(* CODESYS project Elevator - Project Code.project

Project tree, tasks and I/O mapping:
  Device : CODESYS Control Win V3, 3S - Smart Software Solutions GmbH, version 3.5.16.20
    application Application
      libraries: Standard, * (System)
      task MainTask (cyclic, interval t#20ms, priority 1) calls Simulation
      task VISU_TASK (cyclic, interval 100 ms, priority 31) calls VisuElems.Visu_Prg
      global variables GVL
      visualisation Visualization
      program Simulation [ST]
  text list GlobalTextList
*)

// Device/Application/GVL
{attribute 'qualified_only'}
VAR_GLOBAL
(* Elevator managing variables*)
	Open: BOOL;				(* Sensor: the door is fully open*)
	Closed: BOOL;			(* Sensor: the door is fully closed*)
	LimitDown: BOOL;		(* Sensor: lower limit sensor, if TRUE the lift has reached the lower limit*)
	LimitUp: BOOL;			(* Sensor: upper limit sensor, if TRUE the lift has reached the upper limit*)
	DeckSensor: BOOL;		(* Sensor: if TRUE the cab is in proximity of a deck*)
	RampSensor: BOOL;		(* Sensor: if TRUE the cab is in proximity of a ramp*)
	Presence :BOOL; 		(* Sensor: if TRUE something blocks the door photocell*)
	Emergency: BOOL;		(* Input: if TRUE the emergency button has been pressed*)

	Closing: BOOL;			(* Actuator: if TRUE the door starts closing*)
	Opening: BOOL;			(* Actuator: the door starts opening*)
	Motor_on: BOOL;			(* Actuator: if TRUE the lift pulley motor start moving*)
	Up: BOOL;				(* Actuator parameter: if TRUE the lift moves upward, downward otherwise*)
	Vel: BOOL;				(* Actuator parameter: motor speed, if TRUE high speed, low speed otherwise*)


	Current: INT;  			(* Visualization: variable used to storage the current deck*)
    Destination: INT;		(* Visualization: variable used to storage the the destination deck*)
	EmergencyVis: BOOL; 	(* Visualization: if TRUE the emergency light is turned on*)

	InitialDeck: INT := 1;	(* Only for simulation: variable used to define the initial deck*)
	InitCycle: BOOL := FALSE;(* Only for simulation: used to execute the instruction at the first cycle*)
	Height: INT;			(* Only for simulation: elevator height*)
	DeckRest: INT;        	(* Only for simulation: division rest for generating deck sensor*)
	Memory: INT;
	RampRest: INT;			(* Only for simulation: division rest for generating the ramp position*)
	MemoryR: INT;
	Door: INT;				(* Only for simulation: to visualize the closing of the door*)
	Displacement: INT;		(* Only for simulation: lift displacement, dependent on the motor speed*)

 (*Inputs: internal panel variables*)
	PG: BOOL;
	P1: BOOL;
	P2: BOOL;
	P3: BOOL;
	P4: BOOL;
	P5: BOOL;
	P6: BOOL;
	P7: BOOL;

(*Visualization: internal panel variables used to turn on the LED*)
	PGVis: BOOL;
	P1Vis: BOOL;
	P2Vis: BOOL;
	P3Vis: BOOL;
	P4Vis: BOOL;
	P5Vis: BOOL;
	P6Vis: BOOL;
	P7Vis: BOOL;

(*Inputs: external panel variables*)
	UpDeckG: BOOL;
	UpDeck1: BOOL;
	UpDeck2: BOOL;
	UpDeck3: BOOL;
	UpDeck4: BOOL;
	UpDeck5: BOOL;
	UpDeck6: BOOL;
	DownDeck7: BOOL;
	DownDeck6: BOOL;
	DownDeck5: BOOL;
	DownDeck4: BOOL;
	DownDeck3: BOOL;
	DownDeck2: BOOL;
	DownDeck1: BOOL;

(*Visualization: external panel variables used to turn on the LED*)
	UpDeckGVis: BOOL;
	UpDeck1Vis: BOOL;
	UpDeck2Vis: BOOL;
	UpDeck3Vis: BOOL;
	UpDeck4Vis: BOOL;
	UpDeck5Vis: BOOL;
	UpDeck6Vis: BOOL;
	DownDeck7Vis: BOOL;
	DownDeck6Vis: BOOL;
	DownDeck5Vis: BOOL;
	DownDeck4Vis: BOOL;
	DownDeck3Vis: BOOL;
	DownDeck2Vis: BOOL;
	DownDeck1Vis: BOOL;

(*Only for simulation: variables used to simulate the fault on deck sensor*)
	SensorG: BOOL;				(* if TRUE the magnetic information for deck G is lost and the deck sensor cannot become TRUE*)
	Sensor1: BOOL;				(* if TRUE the magnetic information for deck 1 is lost and the deck sensor cannot become TRUE*)
	Sensor2: BOOL;
	Sensor3: BOOL;
	Sensor4: BOOL;
	Sensor5: BOOL;
	Sensor6: BOOL;
	Sensor7: BOOL;
	FaultSensorAlarm: BOOL; 	(* Visulaization: if TRUE alerts the user of a deck sensor fault*)

(*Only for simulation: variables used to simulate the fault on ramp sensor*)
	RampGUp: BOOL;
	Ramp1Down: BOOL;
	Ramp1Up:BOOL;
	Ramp2Down: BOOL;
	Ramp2Up:BOOL;
	Ramp3Down: BOOL;
	Ramp3Up:BOOL;
	Ramp4Down: BOOL;
	Ramp4Up:BOOL;
	Ramp5Down: BOOL;
	Ramp5Up:BOOL;
	Ramp6Down: BOOL;
	Ramp6Up:BOOL;
	Ramp7Down: BOOL;
	FaultRampAlarm: BOOL; 		(* Visulaization: if TRUE alerts the user of a ramp sensor fault*)
	SensorGOK: BOOL;
	Sensor1OK: BOOL;
	Sensor2OK: BOOL;
	Sensor6OK: BOOL;
	Sensor3OK: BOOL;
	Sensor4OK: BOOL;
	Sensor5OK: BOOL;
	Sensor7OK: BOOL;
	RampGUpOK: BOOL;
	Ramp1DownOK: BOOL;
	Ramp1UpOK: BOOL;
	Ramp2DownOK: BOOL;
	Ramp2UpOK: BOOL;
	Ramp3DownOK: BOOL;
	Ramp3UpOK: BOOL;
	Ramp4DownOK: BOOL;
	Ramp4UpOK: BOOL;
	Ramp5DownOK: BOOL;
	Ramp5UpOK: BOOL;
	Ramp6DownOK: BOOL;
	Ramp6UpOK: BOOL;
	Ramp7DownOK: BOOL;
	Ramp7UpOK: BOOL;
END_VAR

// Device/Application/Simulation
PROGRAM Simulation
VAR
END_VAR

(* Initial position of the cab inside the hoistway. It is executed only at the first cycle.  *)
IF NOT GVL.InitCycle THEN
			GVL.InitCycle := TRUE ;
			GVL.Height := 20 * GVL.InitialDeck;
		    GVL.Door := 0;
			GVL.Current := GVL.Height / 20;
END_IF;

(* Elevator management, these instructions are executed each cycle time*)

(* Elevator door control. *)
IF GVL.Closing THEN
	GVL.Door := GVL.Door + 1;		(*Closing door management*)
	GVL.Open := FALSE;
END_IF

IF GVL.Door >= 60 THEN						(* Closed door limit*)
	GVL.Closed := TRUE;
END_IF

IF GVL.Opening THEN
	GVL.Door := GVL.Door - 1; 	(* Opening door management*)
	GVL.Closed := FALSE;
END_IF

IF GVL.Door <= 0 THEN							(* Open door limit*)
	GVL.Open := TRUE;
END_IF


(* Maximum and minimum management in the door simulation*)
IF GVL.Door < 0 THEN
	 GVL.Door := 0;
END_IF

IF GVL.Door > 60 THEN
	GVL.Door := 60;
END_IF


(* Control of the cab position inside the hostway. *)
(* Displacement definition for graphic visualization*)
IF GVL.Vel THEN 
	GVL.Displacement := 2;
ELSE 
	GVL.Displacement := 1;
END_IF


(* Height modification relying on direction and speed*)
IF GVL.Motor_on AND GVL.Up THEN
	GVL.Height := GVL.Height + GVL.Displacement;
	GVL.LimitDown := FALSE;
END_IF

IF GVL.Motor_on AND NOT GVL.Up THEN
	GVL.Height := GVL.Height - GVL.Displacement;
	GVL.LimitUp := FALSE;
END_IF


(* Limits for visualization*)
IF GVL.Height < -20 THEN
	GVL.Height := -20;
END_IF

IF GVL.Height > 160 THEN
	GVL.Height := 160;
END_IF

(* Limit sensors management*)
IF GVL.Height <= -10 THEN
	GVL.LimitDown := TRUE;
END_IF

IF GVL.Height >= 150 THEN
	 GVL.LimitUp := TRUE;
END_IF


(*-------------------------------------------------------------------*)
(*  Fault Management (Deck and Ramp Sensors)   *)
(*-------------------------------------------------------------------*)
(* Deck Sensor*)
(* Range of value where the deck sensor is active*)
IF ((GVL.Height >= -1) AND (GVL.Height <= 1)) THEN
	GVL.SensorGOK := TRUE;
ELSE  
	GVL.SensorGOK := FALSE;
END_IF

IF ((GVL.Height >= 20-1) AND (GVL.Height <= 20+1)) THEN
	GVL.Sensor1OK := TRUE;
ELSE  
	GVL.Sensor1OK := FALSE;
END_IF

IF ((GVL.Height >= 40-1) AND (GVL.Height <= 40+1)) THEN
	GVL.Sensor2OK := TRUE;
ELSE  
	GVL.Sensor2OK := FALSE;
END_IF

IF ((GVL.Height >= 60-1) AND (GVL.Height <= 60+1)) THEN
	GVL.Sensor3OK := TRUE;
ELSE  
	GVL.Sensor3OK := FALSE;
END_IF

IF ((GVL.Height >= 80-1) AND (GVL.Height <= 80+1)) THEN
	GVL.Sensor4OK := TRUE;
ELSE  
	GVL.Sensor4OK := FALSE;
END_IF

IF ((GVL.Height >= 100-1) AND (GVL.Height <= 100+1)) THEN
	GVL.Sensor5OK := TRUE;
ELSE   
	GVL.Sensor5OK := FALSE;
END_IF

IF ((GVL.Height >= 120-1) AND (GVL.Height <= 120+1)) THEN
	GVL.Sensor6OK := TRUE;
ELSE  
	GVL.Sensor6OK := FALSE;
END_IF

IF ((GVL.Height >= 140-1) AND (GVL.Height <= 140+1)) THEN
	GVL.Sensor7OK := TRUE;
ELSE  
	GVL.Sensor7OK := FALSE;
END_IF

GVL.DeckSensor := (GVL.SensorGOK AND NOT GVL.SensorG) OR
				    (GVL.Sensor1OK AND NOT GVL.Sensor1) OR
				    (GVL.Sensor2OK AND NOT GVL.Sensor2) OR
				    (GVL.Sensor3OK AND NOT GVL.Sensor3) OR
				    (GVL.Sensor4OK AND NOT GVL.Sensor4) OR
				    (GVL.Sensor5OK AND NOT GVL.Sensor5) OR
				    (GVL.Sensor6OK AND NOT GVL.Sensor6) OR
				    (GVL.Sensor7OK AND NOT GVL.Sensor7);

(* Ramp Sensor*)
(* Range of value where the ramp sensor is active*)
IF ((GVL.Height >= 5-1) AND (GVL.Height <= 5+1)) THEN
	GVL.RampGUpOK := TRUE;
ELSE 
	GVL.RampGUpOK := FALSE;
END_IF

(* Ramp close to deck 1*)
IF ((GVL.Height >= 15-1) AND (GVL.Height <= 15+1)) THEN
	GVL.Ramp1DownOK := TRUE;
ELSE 
	GVL.Ramp1DownOK := FALSE;
END_IF

IF ((GVL.Height >= 25-1) AND (GVL.Height <= 25+1)) THEN
	GVL.Ramp1UpOK := TRUE;
ELSE 
	GVL.Ramp1UpOK := FALSE;
END_IF

(* Ramp close to deck 2*)
IF ((GVL.Height >= 35-1) AND (GVL.Height <= 35+1)) THEN
	GVL.Ramp2DownOK := TRUE;
ELSE 
	GVL.Ramp2DownOK := FALSE;
END_IF

IF ((GVL.Height >= 45-1) AND (GVL.Height <= 45+1)) THEN
	GVL.Ramp2UpOK := TRUE;
ELSE 
	GVL.Ramp2UpOK := FALSE;
END_IF

(*Ramp close to deck  3*)
IF ((GVL.Height >= 55-1) AND (GVL.Height <= 55+1)) THEN
	GVL.Ramp3DownOK := TRUE;
ELSE 
	GVL.Ramp3DownOK := FALSE;
END_IF

IF ((GVL.Height >= 65-1) AND (GVL.Height <= 65+1)) THEN
	GVL.Ramp3UpOK := TRUE;
ELSE 
	GVL.Ramp3UpOK := FALSE;
END_IF

(* Ramp close to deck  4*)
IF ((GVL.Height >= 75-1) AND (GVL.Height <= 75+1)) THEN
	GVL.Ramp4DownOK := TRUE;
ELSE 
	GVL.Ramp4DownOK := FALSE;
END_IF

IF ((GVL.Height >= 85-1) AND (GVL.Height <= 85+1)) THEN
	GVL.Ramp4UpOK := TRUE;
ELSE 
	GVL.Ramp4UpOK:=FALSE;
END_IF

(* Ramp close to deck  5*)
IF ((GVL.Height >= 95-1) AND (GVL.Height <= 95+1)) THEN
	GVL.Ramp5DownOK := TRUE;
ELSE 
	GVL.Ramp5DownOK := FALSE;
END_IF

IF ((GVL.Height >= 105-1) AND (GVL.Height <= 105+1)) THEN
	GVL.Ramp5UpOK := TRUE;
ELSE
	GVL.Ramp5UpOK := FALSE;
END_IF

(* Ramp close to deck  6*)
IF ((GVL.Height >= 115-1) AND (GVL.Height <= 115+1)) THEN
	GVL.Ramp6DownOK := TRUE;
ELSE 
	GVL.Ramp6DownOK := FALSE;
END_IF

IF ((GVL.Height >= 125-1) AND (GVL.Height <= 125+1)) THEN
	GVL.Ramp6UpOK := TRUE;
ELSE 
	GVL.Ramp6UpOK := FALSE;
END_IF

(* Ramp close to deck  7*)
IF ((GVL.Height >= 135-1) AND (GVL.Height <= 135+1)) THEN
	GVL.Ramp7DownOK := TRUE;
ELSE 
	GVL.Ramp7DownOK := FALSE;
END_IF

GVL.RampSensor:=(GVL.RampGUpOK AND NOT GVL.RampGUp) OR 
								(GVL.Ramp1DownOK AND NOT GVL.Ramp1Down ) OR 
								(GVL.Ramp1UpOK AND NOT GVL.Ramp1Up ) OR
								(GVL.Ramp2DownOK AND NOT GVL.Ramp2Down ) OR 
								(GVL.Ramp2UpOK AND NOT GVL.Ramp2Up ) OR
								(GVL.Ramp3DownOK AND NOT GVL.Ramp3Down ) OR
 								(GVL.Ramp3UpOK AND NOT GVL.Ramp3Up ) OR
								(GVL.Ramp4DownOK AND NOT GVL.Ramp4Down ) OR
 								(GVL.Ramp4UpOK AND NOT GVL.Ramp4Up ) OR
								(GVL.Ramp5DownOK AND NOT GVL.Ramp5Down ) OR
 								(GVL.Ramp5UpOK AND NOT GVL.Ramp5Up ) OR
								(GVL.Ramp6DownOK AND NOT GVL.Ramp6Down ) OR
								(GVL.Ramp6UpOK AND NOT GVL.Ramp6Up ) OR
								(GVL.Ramp7DownOK AND NOT GVL.Ramp7Down );

END_PROGRAM

// Device/Application/Visualization
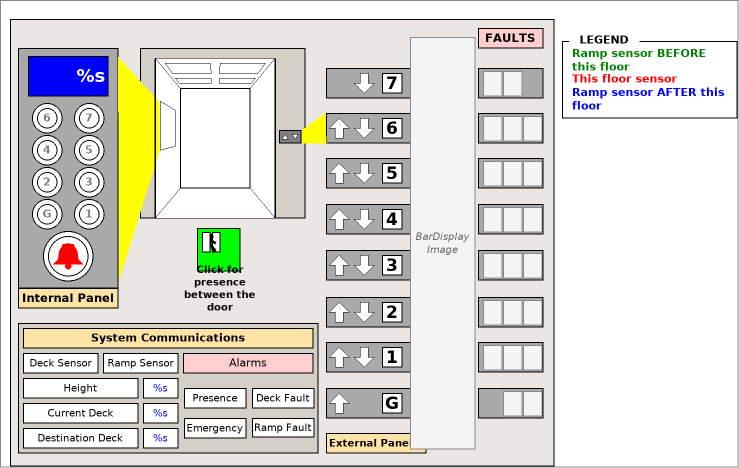
VISUALIZATION Visualization  // 739x468
    Rectangle (10,19 544x447)
    Rectangle (197,228 43x43), colour toggle: GVL.Presence
    Rectangle (18,323 300x130)
    Rectangle (326,433 100x20), "External Panels"
    Rectangle (326,342 100x30)
    Rectangle (382,347 20x20), "1"
    Polygon (354,357) (360,357) (360,347) (368,347) (368,357) (374,357) (364,367), colour toggle: GVL.DownDeck1Vis
        tap GVL.DownDeck1
    Polygon (329,357) (335,357) (335,367) (343,367) (343,357) (349,357) (339,347), colour toggle: GVL.UpDeck1Vis
        tap GVL.UpDeck1
    Rectangle (326,297 100x30)
    Rectangle (382,302 20x20), "2"
    Polygon (354,312) (360,312) (360,302) (368,302) (368,312) (374,312) (364,322), colour toggle: GVL.DownDeck2Vis
        tap GVL.DownDeck2
    Polygon (329,312) (335,312) (335,322) (343,322) (343,312) (349,312) (339,302), colour toggle: GVL.UpDeck2Vis
        tap GVL.UpDeck2
    Rectangle (326,250 100x30)
    Rectangle (382,255 20x20), "3"
    Polygon (354,265) (360,265) (360,255) (368,255) (368,265) (374,265) (364,275), colour toggle: GVL.DownDeck3Vis
        tap GVL.DownDeck3
    Polygon (329,265) (335,265) (335,275) (343,275) (343,265) (349,265) (339,255), colour toggle: GVL.UpDeck3Vis
        tap GVL.UpDeck3
    Rectangle (326,204 100x30)
    Rectangle (382,209 20x20), "4"
    Polygon (354,219) (360,219) (360,209) (368,209) (368,219) (374,219) (364,229), colour toggle: GVL.DownDeck4Vis
        tap GVL.DownDeck4
    Polygon (329,219) (335,219) (335,229) (343,229) (343,219) (349,219) (339,209), colour toggle: GVL.UpDeck4Vis
        tap GVL.UpDeck4
    Rectangle (326,158 100x30)
    Rectangle (382,163 20x20), "5"
    Polygon (354,173) (360,173) (360,163) (368,163) (368,173) (374,173) (364,183), colour toggle: GVL.DownDeck5Vis
        tap GVL.DownDeck5
    Polygon (329,173) (335,173) (335,183) (343,183) (343,173) (349,173) (339,163), colour toggle: GVL.UpDeck5Vis
        tap GVL.UpDeck5
    Rectangle (326,113 100x30)
    Rectangle (382,118 20x20), "6"
    Polygon (354,128) (360,128) (360,118) (368,118) (368,128) (374,128) (364,138), colour toggle: GVL.DownDeck6Vis
        tap GVL.DownDeck6
    Polygon (329,128) (335,128) (335,138) (343,138) (343,128) (349,128) (339,118), colour toggle: GVL.UpDeck6Vis
        tap GVL.UpDeck6
    Rectangle (326,68 100x30)
    Rectangle (382,73 20x20), "7"
    Polygon (354,83) (360,83) (360,73) (368,73) (368,83) (374,83) (364,93), colour toggle: GVL.DownDeck7Vis
        tap GVL.DownDeck7
    Rectangle (326,388 100x30)
    Rectangle (382,393 20x20), "G"
    Polygon (329,403) (335,403) (335,413) (343,413) (343,403) (349,403) (339,393), colour toggle: GVL.UpDeckGVis
        tap GVL.UpDeckG
    RoundedRectangle (18,48 100x240)
    Rectangle (18,288 100x20), "Internal Panel"
    Ellipse (74,199 30x30), colour toggle: GVL.P1Vis
    Ellipse (79,204 20x20), "1"
        tap GVL.P1
    Ellipse (32,199 30x30), colour toggle: GVL.PGVis
    Ellipse (37,204 20x20), "G"
        tap GVL.PG
    Ellipse (74,167 30x30), colour toggle: GVL.P3Vis
    Ellipse (79,172 20x20), "3"
        tap GVL.P3
    Ellipse (32,167 30x30), colour toggle: GVL.P2Vis
    Ellipse (37,172 20x20), "2"
        tap GVL.P2
    Ellipse (74,135 30x30), colour toggle: GVL.P5Vis
    Ellipse (79,140 20x20), "5"
        tap GVL.P5
    Ellipse (32,135 30x30), colour toggle: GVL.P4Vis
    Ellipse (37,140 20x20), "4"
        tap GVL.P4
    Ellipse (74,103 30x30), colour toggle: GVL.P7Vis
    Ellipse (79,108 20x20), "7"
        tap GVL.P7
    Ellipse (32,103 30x30), colour toggle: GVL.P6Vis
    Ellipse (37,108 20x20), "6"
        tap GVL.P6
    Rectangle (28,56 80x40), "%s", text variable: GVL.Destination
    Ellipse (43,231 50x50), tooltip "EMERGENCY", colour toggle: GVL.Emergency
    Group (48,236 40x40)
        toggle GVL.Emergency
        Ellipse (0,0 40x40), tooltip "EMERGENCY"
        Polygon (5,28) (10,23) (11,15) (15,8) (20,7) (25,8) (29,15) (30,23) (35,28)
        Ellipse (17,27 6x6)
    Polygon (35,72) (45,62) (55,72), colour toggle: GVL.Motor_on AND GVL.Up
    Polygon (35,80) (45,90) (55,80), colour toggle: GVL.Motor_on AND NOT GVL.Up
    Group (140,48 165x170)
        Rectangle (0,0 165x170)
        Rectangle (15,10 120x160)
        Polygon (40,40) (15,10) (135,10) (110,40)
        Rectangle (40,40 70x100)
        Polygon (15,170) (40,140) (110,140) (135,170)
        Polygon (20,102) (20,53) (35,62) (35,98)
        Polygon (79,35) (79,30) (115,30) (111,35)
        Polygon (39,35) (35,30) (71,30) (71,35)
        Polygon (32,25) (25,15) (70,15) (71,25)
        Polygon (79,25) (80,15) (125,15) (118,25)
        Group (139,82 22x13)
            Rectangle (0,0 22x13)
            Polygon (3,9) (6,4) (9,9)
            Polygon (13,4) (16,9) (19,4)
    BarDisplayImage (410,37 65x412), value: GVL.Height, style: BarDisplayImage-Gray, scale format: %.0f, scale -20..160
        p3451962224: VisuNativeControl.IP_Offline.Browser
    Rectangle (478,68 65x30)
    Rectangle (478,342 65x30)
    Rectangle (478,297 65x30)
    Rectangle (478,250 65x30)
    Rectangle (478,204 65x30)
    Rectangle (478,158 65x30)
    Rectangle (478,113 65x30)
    Rectangle (478,388 65x30)
    RockerSwitch (483,345 19x25), variable: GVL.Ramp1Down, behaviour: TOGGLE, style: Switch-RockerSwitch-Green
    RockerSwitch (503,345 19x25), variable: GVL.Sensor1, behaviour: TOGGLE, style: Switch-RockerSwitch-Red
    RockerSwitch (523,345 19x25), variable: GVL.Ramp1Up, behaviour: TOGGLE, style: Switch-RockerSwitch-Blue
    RockerSwitch (483,300 19x25), variable: GVL.Ramp2Down, behaviour: TOGGLE, style: Switch-RockerSwitch-Green
    RockerSwitch (503,300 19x25), variable: GVL.Sensor2, behaviour: TOGGLE, style: Switch-RockerSwitch-Red
    RockerSwitch (523,300 19x25), variable: GVL.Ramp2Up, behaviour: TOGGLE, style: Switch-RockerSwitch-Blue
    RockerSwitch (483,253 19x25), variable: GVL.Ramp3Down, behaviour: TOGGLE, style: Switch-RockerSwitch-Green
    RockerSwitch (503,253 19x25), variable: GVL.Sensor3, behaviour: TOGGLE, style: Switch-RockerSwitch-Red
    RockerSwitch (523,253 19x25), variable: GVL.Ramp3Up, behaviour: TOGGLE, style: Switch-RockerSwitch-Blue
    RockerSwitch (483,207 19x25), variable: GVL.Ramp4Down, behaviour: TOGGLE, style: Switch-RockerSwitch-Green
    RockerSwitch (503,207 19x25), variable: GVL.Sensor4, behaviour: TOGGLE, style: Switch-RockerSwitch-Red
    RockerSwitch (523,207 19x25), variable: GVL.Ramp4Up, behaviour: TOGGLE, style: Switch-RockerSwitch-Blue
    RockerSwitch (483,161 19x25), variable: GVL.Ramp5Down, behaviour: TOGGLE, style: Switch-RockerSwitch-Green
    RockerSwitch (503,161 19x25), variable: GVL.Sensor5, behaviour: TOGGLE, style: Switch-RockerSwitch-Red
    RockerSwitch (523,161 19x25), variable: GVL.Ramp5Up, behaviour: TOGGLE, style: Switch-RockerSwitch-Blue
    RockerSwitch (483,116 19x25), variable: GVL.Ramp6Down, behaviour: TOGGLE, style: Switch-RockerSwitch-Green
    RockerSwitch (503,116 19x25), variable: GVL.Sensor6, behaviour: TOGGLE, style: Switch-RockerSwitch-Red
    RockerSwitch (523,116 19x25), variable: GVL.Ramp6Up, behaviour: TOGGLE, style: Switch-RockerSwitch-Blue
    RockerSwitch (483,71 19x25), variable: GVL.Ramp7Down, behaviour: TOGGLE, style: Switch-RockerSwitch-Green
    RockerSwitch (503,71 19x25), variable: GVL.Sensor7, behaviour: TOGGLE, style: Switch-RockerSwitch-Red
    RockerSwitch (503,391 19x25), variable: GVL.SensorG, behaviour: TOGGLE, style: Switch-RockerSwitch-Red
    RockerSwitch (523,391 19x25), variable: GVL.RampGUp, behaviour: TOGGLE, style: Switch-RockerSwitch-Blue
    Rectangle (478,28 65x20), "FAULTS"
    Polygon (302,130) (325,113) (326,143) (302,143), invisible if: (GVL.Closing OR GVL.Opening) OR GVL.Closed
    Polygon (118,57) (159,102) (159,151) (119,279), invisible if: (GVL.Closing OR GVL.Opening) OR GVL.Closed
    Rectangle (155,58 0x160)
        p3528305787: GVL.Door
    Rectangle (275,58 0x160)
        p3528305787: -GVL.Door
    Rectangle (23,328 290x20), "System Communications"
    Rectangle (183,353 130x20), "Alarms"
    Rectangle (23,353 75x20), "Deck Sensor", colour toggle: GVL.DeckSensor
    Rectangle (143,378 35x20), "%s", text variable: GVL.Height
    Rectangle (184,388 62x20), "Presence", colour toggle: GVL.Presence
    Rectangle (103,353 75x20), "Ramp Sensor", colour toggle: GVL.RampSensor
    Rectangle (143,403 35x20), "%s", text variable: GVL.Current
    Rectangle (143,428 35x20), "%s", text variable: GVL.Destination
    Rectangle (252,388 62x20), "Deck Fault", colour toggle: GVL.FaultSensorAlarm
    Rectangle (184,418 62x20), "Emergency", colour toggle: GVL.EmergencyVis
    Rectangle (252,418 62x19), "Ramp Fault", colour toggle: GVL.FaultRampAlarm
    Rectangle (23,378 115x20), "Height"
    Rectangle (23,403 115x20), "Current Deck"
    Rectangle (23,428 115x20), "Destination Deck"
    Group (562,25 175x93)
        Rectangle (0,16 175x77)
        Rectangle (7,39 160x30), "This floor sensor"
        Rectangle (7,59 160x30), "Ramp sensor AFTER this floor"
        Rectangle (7,0 70x30), "LEGEND"
        Rectangle (7,20 160x30), "Ramp sensor BEFORE this floor"
    Group (202,232 33x34)
        toggle GVL.Presence
        Rectangle (10,0 8x20)
        Polygon (5,10) (12,20) (14,18) (5,6)
        Ellipse (6,2 5x5)
        Polygon (4,8) (13,12) (14,10) (4,4)
        Rectangle (0,0 8x20)
    Rectangle (169,273 102x31), "Click for presence between the door"
END_VISUALIZATION
